(* Logix 5000 project; controller R1USB70001_CWRU_GRID_20120217 vendor 1 type 14 code 54 rev 19.11; software revision 19.01; part 2 of 2 *)
(* tags used below, declared in another part *)
   BAT_AC_VOLTAGE : REAL;
   BAT_AC_VOLTAGE_RAW : REAL;
   VOLTAGE_SCALE : REAL;
   BT_GP_ML_ACVT : ALIAS FOR ACNR_GP_SC_N2:9:I.Ch2Data;
   Comment : DINT[2];
(* MainProgram, continued *)

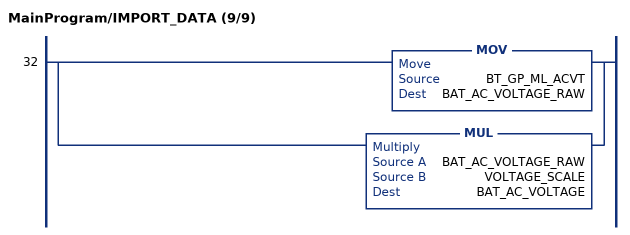
   32: [MOV(BT_GP_ML_ACVT,BAT_AC_VOLTAGE_RAW) ,MUL(BAT_AC_VOLTAGE_RAW,VOLTAGE_SCALE,BAT_AC_VOLTAGE) ];
END_ROUTINE

ROUTINE MainRoutine   (* ladder *)
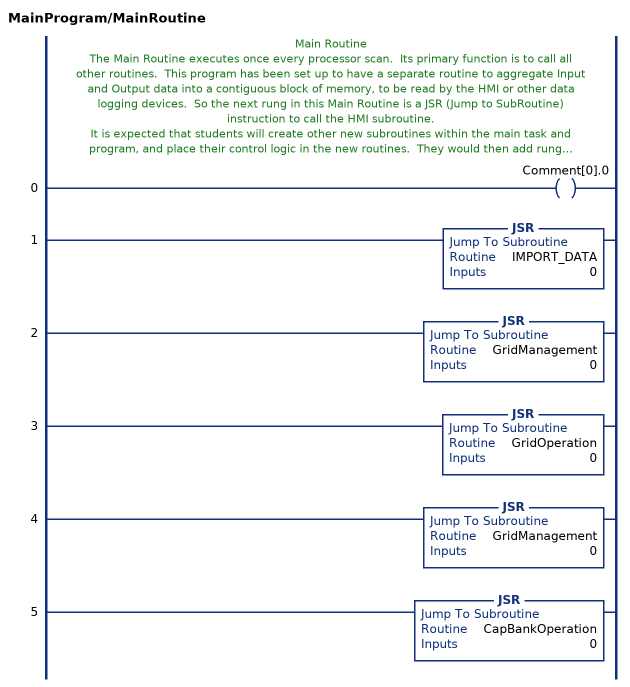
   // Main Routine
   // The Main Routine executes once every processor scan.  Its primary function is to call all other routines.  This program has been set up to have a separate routine to aggregate Input and Output data into a contiguous block of memory, to be read by the HMI or other data logging devices.  So the next rung in this Main Routine is a JSR (Jump to SubRoutine) instruction to call the HMI subroutine.
   // It is expected that students will create other new subroutines within the main task and program, and place their control logic in the new routines.  They would then add rungs within this Main Routine to call the new subroutines that contain their logic.
   0: OTE(Comment[0].0);
   1: JSR(IMPORT_DATA,0);
   2: JSR(GridManagement,0);
   3: JSR(GridOperation,0);
   4: JSR(GridManagement,0);
   5: JSR(CapBankOperation,0);
END_ROUTINE
END_PROGRAM
